{attribute 'qualified_only'}
VAR_GLOBAL
END_VAR

(* stored: Version 1.1.0.1, ProductVersion 3.1.4022.7
   GVL GVL_07_Alarm_Servo_Motor_Shelf_C: Id {f82a6c15-4907-449e-8316-bcc61327c3ac} *)
